// TwinCAT 3 PLC project mqtt_data_gathering
// ProgramVersion: 3.1.4024.0
// libraries:
//   Tc2_Standard, * (Beckhoff Automation GmbH)
//   Tc2_System, * (Beckhoff Automation GmbH)
//   Tc2_Utilities, * (Beckhoff Automation GmbH)
//   Tc3_IotBase, * (Beckhoff Automation GmbH)
//   Tc3_JsonXml, * (Beckhoff Automation GmbH)
//   Tc3_Module, * (Beckhoff Automation GmbH)
// project tree:
//   DUTs/ DevStates.TcDUT, mqtt_data.TcDUT, weather_data.TcDUT
//   GVLs/ GVL.TcGVL
//   / PlcTask.TcTTO
//   POUs/ connect_mqtt.TcPOU, FB_Rest_OpenWeather.TcPOU, location_PushBack.TcPOU, MAIN.TcPOU, setup_mqtt.TcPOU
// real-time tasks:
//   TASK PlcTask: cycle T#10ms, priority 20, ADS port 350

CONFIGURATION mqtt_data_gathering
    RESOURCE PLC ON TwinCAT3
        TASK PlcTask(INTERVAL := T#10ms, PRIORITY := 20);
        PROGRAM MAIN WITH PlcTask : MAIN;
    END_RESOURCE
END_CONFIGURATION

// ---- DUTs/DevStates.TcDUT
{attribute 'qualified_only'}
{attribute 'strict'}
TYPE DevStates :
(
	NOOP := 0,
	IDLE,
 	RECEIVING,
	PROC,
	SENDING,
	ERR
);
END_TYPE

// ---- DUTs/mqtt_data.TcDUT
TYPE mqtt_data :
STRUCT
	fbMqttClient : FB_IotMqttClient;
	bSetParameter : BOOL := TRUE;
	bConnect : BOOL := TRUE;
	
	(* published message *)
	sTopicPub : STRING(255) := 'testtopic/out';
	sPayloadPub : STRING(255);
	
	
	(* received message *)
	bSubscribed : BOOL;
	sTopicSub : STRING(255) := 'testtopic/in';
	{attribute 'TcEncoding':='UTF-8'}
	sTopicRcv : STRING(255);
	{attribute 'TcEncoding':='UTF-8'}
	sPayloadRcv : STRING(255);
	fbMessageQueue : FB_IotMqttMessageQueue;
	fbMessage : FB_IotMqttMessage;
	
	hrErrorOccurred : HRESULT; // contains the latest occurred error
	btimeout: BOOL;
END_STRUCT
END_TYPE

// ---- DUTs/weather_data.TcDUT
TYPE weather_data :
STRUCT
	student_id  : DINT := 12202053; 
	last        : STRING(64) := 'jaworski';
   	first       : STRING(64) := 'oliwier';
    sLocation 	: ARRAY[1..4] OF STRING(255);
	
	city      	: STRING(64);
    id          : UDINT;
    temp        : LREAL;
    temp_min    : FLOAT;
    temp_max    : FLOAT;
    sunrise     : UDINT;
    sunset      : UDINT;
	
	uLocIndex		: UINT :=0;
    sJsonParsed     : STRING(2048);
	
	allow_processing : BOOL := FALSE;
END_STRUCT
END_TYPE

// ---- GVLs/GVL.TcGVL
{attribute 'qualified_only'}
VAR_GLOBAL
	MAX_SIZE : UINT := 4;
END_VAR

// ---- POUs/MAIN.TcPOU
PROGRAM MAIN
VAR
	btimeout 		: BOOL;
	sState 			: DevStates;
	M_data			: mqtt_data;
	W_data 			: weather_data;
	fbMqttClient: INT;
	fbMessageQueue: INT;
	fbTimer : TON := (PT:=T#10S);
	refMqtt: INT;
	Execute: INT;
	
	bGetOpenWeatherMap 				: BOOL; 

	fbHttpClientOpenWeatherMap		: FB_IotHttpClient :=(sHostName := 'api.openweathermap.org',
								  	bKeepAlive := TRUE,	tConnectionTimeout := T#10S);

	fbHttpGetOpenWeatherMap			: FB_Rest_OpenWeather;
	
	fbJsonSAX 						: FB_JsonSaxWriter;
	bSAXheader						: BOOL :=FALSE;
END_VAR

(* ERROR HANDLING*)
IF sState = DevStates.ERR THEN
	// Very high level error handling will happen here
END_IF

(* PROCESS MEMBER SETUP *)
IF sState = DevStates.NOOP THEN
	sState := setup_mqtt(refMqtt := M_data, refUser := W_data, refState := sState);
	sState := DevStates.RECEIVING;
END_IF

(* FETCH DATA UNTIL TIMEOUT *)
IF sState = DevStates.RECEIVING THEN
	connect_mqtt(M_data := M_data);
	IF  W_data.uLocIndex <> 0  THEN
		//only start the timer if some data has been received and waiting for timeout
		fbTimer(IN:=TRUE);
	END_IF
	
	IF M_data.fbMessageQueue.nQueuedMessages > 0 THEN
		IF M_data.fbMessageQueue.Dequeue(fbMessage:=M_data.fbMessage) THEN
			M_data.fbMessage.GetTopic(pTopic:=ADR(M_data.sTopicRcv), nTopicSize:=SIZEOF(M_data.sTopicRcv) );
			M_data.fbMessage.GetPayload(pPayload:=ADR(M_data.sPayloadRcv), nPayloadSize:=SIZEOF(M_data.sPayloadRcv), bSetNullTermination:=TRUE);
			IF  W_data.uLocIndex <= GVL.MAX_SIZE  THEN
                location_PushBack(refdata := W_data, refinput := M_data.sPayloadRcv);
				fbTimer(IN := FALSE);
			END_IF;
		END_IF
	END_IF
	IF fbTimer.Q THEN
		//get value from string and push back into array.
		fbTimer(IN:=FALSE);
		sState := DevStates.PROC;
	END_IF
END_IF

(* FETCH DATA FROM OPENWEATHER *)
IF sState = DevStates.PROC THEN
	IF NOT bSAXheader THEN
		fbJsonSAX.StartObject();
		fbJsonSAX.AddKey('user');
			fbJsonSAX.StartObject();
				fbJsonSAX.AddKey('id');
				fbJsonSAX.AddDint(W_data.student_id);
				fbJsonSAX.AddKey('last');
				fbJsonSAX.AddString(W_data.last);
				fbJsonSAX.AddKey('first');
				fbJsonSAX.AddString(W_data.first);
			fbJsonSAX.EndObject();
			fbJsonSAX.AddKey('weather');
			fbJsonSAX.StartArray(); 
			bSAXheader := TRUE;
	END_IF
	
	IF NOT fbHttpClientOpenWeatherMap.bConfigured THEN 
		fbHttpClientOpenWeatherMap.nHostPort := 443;
		fbHttpClientOpenWeatherMap.stTLS.bNoServerCertCheck := TRUE;
	END_IF
	
	
	IF W_data.uLocIndex > 0 THEN
		bGetOpenWeatherMap := TRUE;
		IF fbHttpClientOpenWeatherMap.bConfigured THEN
		fbHttpGetOpenWeatherMap(bSend := bGetOpenWeatherMap, fbClient := fbHttpClientOpenWeatherMap, refState := sState, W_data := W_data);
		END_IF
		fbHttpClientOpenWeatherMap.Execute();
		IF W_data.allow_processing <> FALSE THEN
			fbJsonSAX.StartObject();
				fbJsonSAX.AddKey('city');
				fbJsonSAX.AddString(W_data.city);
				fbJsonSAX.AddKey('id');
				fbJsonSAX.AddUdint(W_data.id);
				fbJsonSAX.AddKey('temp');
				fbJsonSAX.AddLreal(W_data.temp);
				fbJsonSAX.AddKey('temp_min');
				fbJsonSAX.AddLreal(W_data.temp_min);
				fbJsonSAX.AddKey('temp_max');
				fbJsonSAX.AddLreal(W_data.temp_max);
				fbJsonSAX.AddKey('sunrise');
				fbJsonSAX.AddUdint(W_data.sunrise);
				fbJsonSAX.AddKey('sunset');
				fbJsonSAX.AddUdint(W_data.sunset);
				fbJsonSAX.EndObject();
			W_data.allow_processing := FALSE;
			W_data.uLocIndex := W_data.uLocIndex -1;
		END_IF
	ELSE
		fbJsonSAX.EndArray(); 
		fbJsonSAX.EndObject();
		W_data.sJsonParsed := fbJsonSAX.GetDocument();
		fbJsonSAX.CopyDocument(W_data.sJsonParsed, SIZEOF(W_data.sJsonParsed));
		sState := DevStates.SENDING;
	END_IF
	
END_IF

(* SEND RESULTING JSON OBJECT *)
IF sState = DevStates.SENDING THEN
	W_data.uLocIndex := 0;(* FLUSH ARRAY *)
	connect_mqtt(M_data := M_data);
	//sPayloadPub := CONCAT('MyMessage', TO_STRING(i));
		M_data.fbMqttClient.Publish(	sTopic:= M_data.sTopicPub, 
								pPayload:= ADR(W_data.sJsonParsed), nPayloadSize:= LEN(W_data.sJsonParsed)+1, 
								eQoS:= TcIotMqttQos.AtMostOnceDelivery, bRetain:= FALSE, bQueue:= FALSE );
		IF M_data.fbMqttClient.bError THEN
			// add your error logging here
			M_data.hrErrorOccurred := M_data.fbMqttClient.hrErrorCode;
		END_IF
		sState := DevStates.RECEIVING;
END_IF


IF sState = DevStates.IDLE THEN
	(* WASTE TIME *)
END_IF

END_PROGRAM

// ---- POUs/FB_Rest_OpenWeather.TcPOU
FUNCTION_BLOCK FB_Rest_OpenWeather
VAR_INPUT
	bSend				: BOOL;
	refState 			: REFERENCE TO DevStates;
	W_data 			 	: REFERENCE TO weather_data;
END_VAR
VAR_IN_OUT    	
	fbClient			: FB_IotHttpClient;
END_VAR
VAR_OUTPUT
	bBusy				: BOOL;
	bError				: BOOL;
END_VAR
VAR
	fbRequest			: FB_IotHttpRequest;
	fbJson				: FB_JsonDomParser;
	nState				: UDINT;
	RisingEdge			: R_TRIG;
	
	bGetContentResult	: BOOL;
	sContent			: STRING(1023);	
	stest				: STRING(1023) := '{"coord":{"lon":5.3378,"lat":50.9311},"weather":[{"id":804,"main":"Clouds","description":"overcast clouds","icon":"04n"}],"base":"stations","main":{"temp":286.8,"feels_like":286.57,"temp_min":286.16,"temp_max":287.03,"pressure":1025,"humidity":90,"sea_level":1025,"grnd_level":1018},"visibility":10000,"wind":{"speed":2.59,"deg":238,"gust":5.48},"clouds":{"all":89},"dt":1759799774,"sys":{"type":1,"id":1230,"country":"BE","sunrise":1759816113,"sunset":1759856646},"timezone":7200,"id":2796491,"name":"Hasselt","cod":200}';
	bGetJsonResult		: BOOL;
	jsonDoc				: SJsonValue;
	jsonVal				: SJsonValue;
	fResultValue		: LREAL;
	
	nReqCount			: UDINT;	
	nResCount			: UDINT;
	nValidResCount		: UDINT;
	nErrCount			: UDINT;
	
	(* JSON SPECIFIC*)
	nCount  : UDINT;
	idx     : UDINT;
    jsonObj     : SJsonValue;	
	
	sUri        : STRING(256);
	key        : STRING(256) :='';
END_VAR

RisingEdge(CLK := bSend);

CASE nState OF
3:
	jsonDoc := fbJson.ParseDocument(stest);
    IF jsonDoc <> 0 THEN
		// --- city name ---
		IF fbJson.HasMember(jsonDoc, 'name') THEN
			jsonObj := fbJson.FindMember(jsonDoc, 'name');
			W_data.city := fbJson.GetString(jsonObj);
		END_IF;
	
		// --- city id ---
		IF fbJson.HasMember(jsonDoc, 'id') THEN
			W_data.id := fbJson.GetUint(fbJson.FindMember(jsonDoc, 'id')); // numeric type = LREAL, cast ok
		END_IF;
	
		// --- main temperatures ---
		IF fbJson.HasMember(jsonDoc, 'main') THEN
			jsonObj := fbJson.FindMember(jsonDoc, 'main');
			W_data.temp     := fbJson.GetDouble(fbJson.FindMember(jsonObj, 'temp'));
			W_data.temp_min := fbJson.GetDouble(fbJson.FindMember(jsonObj, 'temp_min'));
			W_data.temp_max := fbJson.GetDouble(fbJson.FindMember(jsonObj, 'temp_max'));
		END_IF;
	
		// --- sys (sunrise/sunset) ---
		IF fbJson.HasMember(jsonDoc, 'sys') THEN
			jsonObj := fbJson.FindMember(jsonDoc, 'sys');
			W_data.sunrise := fbJson.GetUint(fbJson.FindMember(jsonObj, 'sunrise'));
			W_data.sunset  := fbJson.GetUint(fbJson.FindMember(jsonObj, 'sunset'));
		END_IF;
	END_IF
	
	W_data.allow_processing := TRUE;
	
		
0:	
	IF RisingEdge.Q THEN 
		sUri := '/data/2.5/weather?q=';
		sUri := CONCAT(sUri, W_data.sLocation[W_data.uLocIndex]);
		sUri := CONCAT(sUri, '&limit=1&appid=');
		sUri := CONCAT(sUri, key);
		IF fbRequest.SendRequest(sUri := sUri, fbClient := fbClient, eRequestType := ETcIotHttpRequestType.HTTP_GET, 0, 0, 0) THEN				
			nState := 1;
			nReqCount := nReqCount +1;
			bBusy := TRUE;
			bError := FALSE;
			bSend := FALSE;
		END_IF					
	END_IF
1:
	IF NOT fbRequest.bBusy THEN
		bError := TRUE;
		IF NOT fbRequest.bError THEN				 
			// As an alternative to GetJsonDomContent, GetContent could be used				 
			// bGetContentResult := fbRequest.GetContent(pContent := ADR(sContent), nContentSize := SIZEOF(sContent), bSetNullTermination := TRUE);
			IF fbRequest.nStatusCode >= 200 AND fbRequest.nStatusCode < 300 THEN
				bGetJsonResult := FALSE;
				// Direct conversion into JSON object as the received message is in JSON format 
				jsonDoc := fbRequest.GetJsonDomContent(fbJson);
							//idk do something	json parsing will go here
				//jsonDoc := fbJson.ParseDocument(stest);
			
				IF jsonDoc <> 0 THEN
					// --- city name ---
					IF fbJson.HasMember(jsonDoc, 'name') THEN
						jsonObj := fbJson.FindMember(jsonDoc, 'name');
						W_data.city := fbJson.GetString(jsonObj);
					END_IF;
				
					// --- city id ---
					IF fbJson.HasMember(jsonDoc, 'id') THEN
						W_data.id := fbJson.GetUint(fbJson.FindMember(jsonDoc, 'id')); // numeric type = LREAL, cast ok
					END_IF;
				
					// --- main temperatures ---
					IF fbJson.HasMember(jsonDoc, 'main') THEN
						jsonObj := fbJson.FindMember(jsonDoc, 'main');
						W_data.temp     := fbJson.GetDouble(fbJson.FindMember(jsonObj, 'temp'));
						W_data.temp_min := fbJson.GetDouble(fbJson.FindMember(jsonObj, 'temp_min'));
						W_data.temp_max := fbJson.GetDouble(fbJson.FindMember(jsonObj, 'temp_max'));
					END_IF;
				
					// --- sys (sunrise/sunset) ---
					IF fbJson.HasMember(jsonDoc, 'sys') THEN
						jsonObj := fbJson.FindMember(jsonDoc, 'sys');
						W_data.sunrise := fbJson.GetUint(fbJson.FindMember(jsonObj, 'sunrise'));
						W_data.sunset  := fbJson.GetUint(fbJson.FindMember(jsonObj, 'sunset'));
					END_IF;
				END_IF
				
				W_data.allow_processing := TRUE;	
				
				END_IF							
				nResCount := nResCount +1;			
			nState := 0;
			bBusy := FALSE;
			IF bError THEN
				nErrCount := nErrCount +1;
			END_IF
		//refState := DevStates.SENDING;
		END_IF
	END_IF   	
END_CASE

END_FUNCTION_BLOCK

// ---- POUs/setup_mqtt.TcPOU
FUNCTION setup_mqtt : DevStates
VAR_INPUT
	refUser : REFERENCE TO weather_data;
	refMqtt : REFERENCE TO mqtt_data;
	refState: REFERENCE TO DevStates;
END_VAR
VAR_OUTPUT
	out : DevStates;
END_VAR
VAR
END_VAR

refMqtt.bSetParameter := FALSE;
refMqtt.fbMqttClient.sHostName:= '3af27b0972ae4f52a828b3b86b9213d0.s1.eu.hivemq.cloud';
refMqtt.fbMqttClient.nHostPort:= 8883;
refMqtt.fbMqttClient.sClientId:= 'test_user';
refMqtt.fbMqttClient.sUserName:= 'test_user';
refMqtt.fbMqttClient.sUserPassword:= 'Test_user01!'; 
refMqtt.fbMqttClient.nKeepAlive:= 60;
refMqtt.fbMqttClient.sTopicPrefix:= ''; 
refMqtt.fbMqttClient.stTLS.bNoServerCertCheck :=  TRUE;
refMqtt.fbMqttClient.ipMessageQueue := refMqtt.fbMessageQueue;

END_FUNCTION

// ---- POUs/connect_mqtt.TcPOU
FUNCTION connect_mqtt : DevStates
VAR_INPUT
	M_data : REFERENCE TO mqtt_data;
END_VAR
VAR
END_VAR

M_data.fbMqttClient.Execute(M_data.bConnect);
IF M_data.fbMqttClient.bError THEN
	// add your error logging here
	M_data.hrErrorOccurred := M_data.fbMqttClient.hrErrorCode;
	connect_mqtt :=  DevStates.ERR;
	RETURN;
END_IF

IF M_data.fbMqttClient.bConnected THEN
	IF NOT M_data.bSubscribed THEN
		M_data.bSubscribed := M_data.fbMqttClient.Subscribe(sTopic:=M_data.sTopicSub, eQoS:=TcIotMqttQos.AtMostOnceDelivery);
		IF M_data.fbMqttClient.bError THEN
			// add your error logging here
			M_data.hrErrorOccurred := M_data.fbMqttClient.hrErrorCode;
			connect_mqtt :=  DevStates.ERR;
			RETURN;
		END_IF
		connect_mqtt := DevStates.RECEIVING;
	END_IF
END_IF

END_FUNCTION

// ---- POUs/location_PushBack.TcPOU
FUNCTION location_PushBack : string
VAR_INPUT
	refdata : REFERENCE TO weather_data;
	refinput : REFERENCE TO STRING;
END_VAR
VAR
    nCommaPos : INT;
    nLen      : INT;
END_VAR

(* FUNC checks if provided string format is correct.*)
nCommaPos := FIND(refinput, ','); // returns 0 if not found
IF nCommaPos = 0 THEN
    RETURN;
END_IF

// Check length after comma
nLen := LEN(refinput);
IF (nLen - nCommaPos) = 2 THEN
	refdata.uLocIndex :=  refdata.uLocIndex + 1;
    refdata.sLocation[refdata.uLocIndex] := refinput;
END_IF

END_FUNCTION
